VAR_GLOBAL CONSTANT
	MAX_D_OUT	: INT := 1;
END_VAR

(* stored: Version 1.1.0.1, ProductVersion 3.1.0.36
   GVL IO_DigiOut_Parameters: Id {d680a340-89e2-43da-8ce1-394be3fad291}, ParameterList True *)
